FUNCTION_BLOCK PtInterval IMPLEMENTS I_PtInterval
VAR_INPUT
END_VAR
VAR_OUTPUT
END_VAR
VAR
	_Start : PtDateTime;
	_End : PtDateTime;
	_Absolute : BOOL;
	
	_DeltaYears : DINT;
	_DeltaMonths : DINT;
	_DeltaDays : DINT;
END_VAR

PROPERTY Absolute : BOOL
GET
Absolute := _Absolute;
END_GET
SET
_Absolute := Absolute;
END_SET
END_PROPERTY

PROPERTY End : PtDateTime
GET
End := _End;
END_GET
SET
_End := End;
END_SET
END_PROPERTY

METHOD inMonth : DINT
VAR_INPUT
END_VAR
inMonth := ABS(_Start.Month - _End.Month);
END_METHOD

METHOD inYears : DINT
VAR_INPUT
END_VAR
inYears := ABS(_Start.Year - _End.Year);
END_METHOD

METHOD Set //: BOOL
VAR_INPUT
	Start : PtDateTime;
	End : PtDateTime;
	Absolute : BOOL;
END_VAR
_Start := Start;
_End := End;
_Absolute := Absolute;

_DeltaYears := ABS(_Start.Year - _End.Year);
_DeltaMonths := ABS(_Start.Month - _End.Month);
_DeltaDays := ABS(_Start.Day - End.Day);
END_METHOD

PROPERTY Start : PtDateTime
GET
END_GET
SET
_Start := Start;
END_SET
END_PROPERTY

END_FUNCTION_BLOCK

(* stored: Version 1.1.0.1, ProductVersion 3.1.4024.12
   POU PtInterval: Id {6c220e54-6a7d-4c45-b8b4-392958277534}, SpecialFunc None
   Property Absolute: Id {fec456c7-312c-4182-9f81-52f94949c278}
   Get Get: Id {f94b6dae-7d0e-4849-9658-4e72bc92e150}
   Set Set: Id {4effa8a0-5a47-43b0-bc16-31a1d4f8c28e}
   Property End: Id {7f96099d-836c-455f-9a36-1dd9612175f4}
   Get Get: Id {03abbfb9-0141-444d-b64b-8c2c8f23dfd3}
   Set Set: Id {85d069e0-bcfb-47b1-847e-a0ac7d44ae23}
   Method inMonth: Id {3f805b12-77c8-4efa-981a-1c359310ea3c}
   Method inYears: Id {05ca97f9-3476-4da7-9f14-f56c00052842}
   Method Set: Id {e1529dd6-6f54-4f80-a00b-cbab76f60ec7}
   Property Start: Id {b97f8927-5eba-4762-8baf-031c94c1d060}
   Get Get: Id {9a74b41a-a93b-42d0-aa5b-2229d79a2c23}
   Set Set: Id {d026f405-9b54-42da-9ae8-e8999ad3f402} *)
